Fanuc KAREL source: READ_DICT.kl

PROGRAM T
%NOLOCKGROUP
VAR
 v0 : STRING[40]
 v1 : INTEGER
 v2 : ARRAY[10] OF STRING[40]
 v3 : INTEGER
 v4 : INTEGER
 v5 : INTEGER
BEGIN
 READ_DICT(v0, v1, v2, v3, v4, v5)
END T
